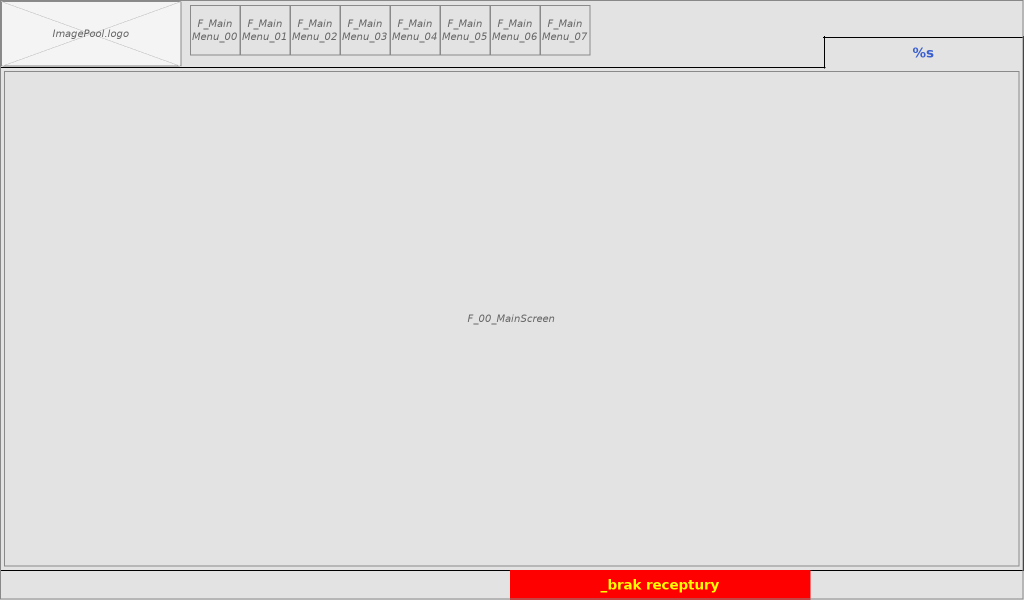
VISUALIZATION MainFrame  // 1024x600
VAR_IN_OUT
	stHMIData		: ST_HMIManager;
END_VAR
    Image (1,1 180x65), image: ImagePool.logo
    Frame (190,5 50x50)
        shows F_MainMenu_00(stMenuButton := stHMIData.stMainMenu.arrButton [0].stButtonHMI)
    Frame (240,5 50x50)
        shows F_MainMenu_01(stMenuButton := stHMIData.stMainMenu.arrButton [1].stButtonHMI)
    Frame (290,5 50x50)
        shows F_MainMenu_02(stMenuButton := stHMIData.stMainMenu.arrButton [2].stButtonHMI)
    Frame (340,5 50x50)
        shows F_MainMenu_03(stMenuButton := stHMIData.stMainMenu.arrButton [3].stButtonHMI)
    Frame (390,5 50x50)
        shows F_MainMenu_04(stMenuButton := stHMIData.stMainMenu.arrButton [4].stButtonHMI)
    Frame (440,5 50x50)
        shows F_MainMenu_05(stMenuButton := stHMIData.stMainMenu.arrButton [5].stButtonHMI)
    Frame (490,5 50x50)
        shows F_MainMenu_06(stMenuButton := stHMIData.stMainMenu.arrButton [6].stButtonHMI)
    Frame (540,5 50x50)
        shows F_MainMenu_07(stMenuButton := stHMIData.stMainMenu.arrButton [7].stButtonHMI)
    Line (0,67) (825,67)
    Line (824,36) (824,68)
    Line (1023,36) (1023,570)
    Line (823,37) (1024,37)
    Line (0,570) (1024,570)
    Line (0,67) (0,570)
    Rectangle (510,570 300x30), "_brak receptury", text list: 'TextList_Ekran', text index: 18
    Rectangle (827,40 193x26), "%s", text variable: stHMIData.stMainMenu.stMenu.wsTitleActivePage
    Frame (4,71 1015x495), frame switch variable: stHMIData.stMainMenu.stMenu.iNumberOfActivePage
        shows F_00_MainScreen()
        shows F_01_Parameters(stScreenData := stHMIData.stMachineControl.stPrepScr_01_XX)
        shows F_02_Recipe(stScreenData := stHMIData.stMachineControl.stPrepScr_02_XX)
        shows F_03_Events(stScreenData := stHMIData.stMachineControl.stPrepScr_03_XX)
        shows F_04_ChangeMode(stScreenData := stHMIData.stMachineControl.stPrepScr_04_XX)
        shows F_05_Statistics(stScreenData := stHMIData.stMachineControl.stPrepScr_05_XX)
        shows F_06_Diagram(stScreenData := stHMIData.stMachineControl.stPrepScr_06_XX)
        shows F_07_Settings(stScreenData := stHMIData.stMachineControl.stPrepScr_07_XX)
END_VISUALIZATION

(* stored: Version 1.1.0.1
   Visu MainFrame: Id {5e796c2a-108a-4a22-84c5-51a3c221ec40} *)
